KUKA KRL program: ChillerOn.src

&ACCESS RVO2
&REL 49
&PARAM EDITMASK = *
&PARAM TEMPLATE = C:\KRC\Roboter\Template\vorgabe
DEF ChillerOn( )

;************************************************
;              CNC Robotics Ltd
;              www.cncrobotics.co.uk
;************************************************
;     Contact: helpdesk@cncrobotics.co.uk
;     Date: 25/09/23
;     Version: 0.14.46
;************************************************
; Description: Routine to turn on the spindle
;************************************************
bRequestChiller = TRUE
WAIT FOR oCoolantOn
WAIT FOR iChillerRunning
bChillerRunning=TRUE
END
